(* CODESYS project cliamat_241cec24t.project
   CustomField05_name: CustomField05
   CustomField06_name: CustomField06
   CustomField08_name: CustomField08
   Version: 1.0.0.0
   CustomField04_name: CustomField04
   Company: Entel & ZIT
   CustomField07_name: CustomField07
   CustomField09_name: CustomField09
   CustomField02_name: CustomField02
   Title: Skrebka climat
   Description: This template can be used for a correct interface with the local drive. the MANDATORY_AT_EACH_CYCLE program must be called like it is done in this application.
   CustomField01_name: CustomField01
   CustomField03_name: CustomField03
   CustomField10_name: CustomField10

Project tree, tasks and I/O mapping:
  MyController : TM241CEC24T/U, Schneider Electric, order no. TM241CEC24T/U, version 4.0.2.20
    application Application
      task MAST (cyclic, interval 20 ms, priority 15, watchdog 100 ms x 1) calls MyPOU, Alarm_checker
      function HiddenPOU [ST]
      global variables GVL
      program MyPOU [ST]
      data type CLIMAT_STATE
      program Alarm_checker [ST]
      data type ON_OFF_STATE
      data type OUT_VENTILATION_STATE
      Relocation Table
    DQ : Digital Outputs, Schneider Electric, version 4.0.2.20
        output qbDQ_QB1 : BYTE  // QB1
        unmapped channels: QW0
    Counters : Counters, Schneider Electric, version 4.0.2.20
    Pulse_Generators : Pulse Generators, Schneider Electric, version 4.0.2.20
    Cartridge_1 : Cartridge, Schneider Electric, version 4.0.2.20
    IO_Bus : IO bus - TM3, Schneider Electric, version 4.0.2.20
      Digital_Ouput_Module : TM3DQ16R/G, Schneider Electric, order no. TM3DQ16R/G, version 1.0.1.2
          output ctr_fans : BOOL  // QW0.Q0
          output ctr_heating : BOOL  // QW0.Q1
          output ctr_vent_valves : BOOL  // QW0.Q2
          output ctr_recirc_valves : BOOL  // QW0.Q3
          output ctr_devices_heating : BOOL  // QW0.Q4
          output ctr_call_staff : BOOL  // QW0.Q8
          output ctr_alarm : BOOL  // QW0.Q9
          unmapped channels: QW0
      Analog_Input_Module : TM3TI8T/G, Schneider Electric, order no. TM3TI8T/G, version 1.0.1.6
          settings: KPI Configuration.KPI Configuration[0] = 73; KPI Configuration.KPI Configuration[1] = 73; KPI Configuration.KPI Configuration[2] = 73; KPI Configuration.KPI Configuration[3] = 73; KPI Configuration.KPI Configuration[8] = 48; KPI Configuration.KPI Configuration[9] = 248; KPI Configuration.KPI Configuration[10] = 48; KPI Configuration.KPI Configuration[11] = 248; KPI Configuration.KPI Configuration[12] = 48; KPI Configuration.KPI Configuration[13] = 248; KPI Configuration.KPI Configuration[14] = 48; KPI Configuration.KPI Configuration[15] = 248; KPI Configuration.KPI Configuration[24] = 64; KPI Configuration.KPI Configuration[25] = 31; KPI Configuration.KPI Configuration[26] = 64; KPI Configuration.KPI Configuration[27] = 31; KPI Configuration.KPI Configuration[28] = 64; KPI Configuration.KPI Configuration[29] = 31; KPI Configuration.KPI Configuration[30] = 64; KPI Configuration.KPI Configuration[31] = 31
          input  temp_in_raw : INT  // IW0
          input  temp_exhaust_raw : INT  // IW1
          input  temp_out_raw : INT  // IW2
          input  temp_supply_raw : INT  // IW3
          input  ibModule_3_IBStatusIW0 : BYTE  // IBStatusIW0
          input  ibModule_3_IBStatusIW1 : BYTE  // IBStatusIW1
          input  ibModule_3_IBStatusIW2 : BYTE  // IBStatusIW2
          input  ibModule_3_IBStatusIW3 : BYTE  // IBStatusIW3
          input  ibModule_3_IBStatusIW4 : BYTE  // IBStatusIW4
          input  ibModule_3_IBStatusIW5 : BYTE  // IBStatusIW5
          input  ibModule_3_IBStatusIW6 : BYTE  // IBStatusIW6
          input  ibModule_3_IBStatusIW7 : BYTE  // IBStatusIW7
          unmapped channels: IW4, IW5, IW6, IW7
      Analog_Output_Module : TM3AQ2/G, Schneider Electric, order no. TM3AQ2/G, version 1.0.0.10
          settings: KPI Configuration.KPI Configuration[0] = 16; KPI Configuration.KPI Configuration[1] = 16; KPI Configuration.KPI Configuration[3] = 0; KPI Configuration.KPI Configuration[5] = 0; KPI Configuration.KPI Configuration[6] = 16; KPI Configuration.KPI Configuration[7] = 39; KPI Configuration.KPI Configuration[8] = 16; KPI Configuration.KPI Configuration[9] = 39
          output fan_speed : INT  // QW0
          input  ibModule_4_IBStatusQW0 : BYTE  // IBStatusQW0
          input  ibModule_4_IBStatusQW1 : BYTE  // IBStatusQW1
          unmapped channels: QW1
    COM_Bus : COM bus, Schneider Electric, version 4.0.2.20
    Serial_Line_2 : Serial line, Schneider Electric, version 4.0.2.20
      Modbus_Manager : Modbus Manager, Schneider Electric, version 4.0.0.2
    CAN_1 : CANopen bus, Schneider Electric, version 4.0.2.20
    DI : Digital Inputs, Schneider Electric, version 4.0.2.20
        input  Application.MyPOU.input_raw : WORD  // IW0
        input  is_fan_exhauster : BOOL  // IW0.I0
        input  is_fan_supply : BOOL  // IW0.I1
        input  is_heating : BOOL  // IW0.I2
        input  is_vent_valves : BOOL  // IW0.I3
        input  is_recirc_valves : BOOL  // IW0.I4
        input  is_devices_heating : BOOL  // IW0.I5
        input  is_on_automation : BOOL  // IW0.I6
        input  is_alarm_fire : BOOL  // IW0.I8
        input  is_alarm_no_voltage_raw : BOOL  // IW0.I9
        input  is_alarm_clogging_1 : BOOL  // IW0.I10
        input  is_alarm_clogging_2 : BOOL  // IW0.I11
        input  ibDI_IB1 : BYTE  // IB1
    Ethernet_1 : Ethernet Network, Schneider Electric, version 4.0.2.20
    Serial_Line_1 : Serial line, Schneider Electric, version 4.0.2.20
      Modbus_Manager_Out : Modbus Manager, Schneider Electric, version 4.0.0.2
*)

// MyController/Application/CLIMAT_STATE
TYPE CLIMAT_STATE :
(
	NORMAL := 0,
	HEATING,
	CRITICAL_HEATING
);
END_TYPE

// MyController/Application/ON_OFF_STATE
TYPE ON_OFF_STATE :
(
	STATE_ON := 0,
	STATE_OFF
);
END_TYPE

// MyController/Application/OUT_VENTILATION_STATE
TYPE OUT_VENTILATION_STATE :
(
	OUT_VENT_NORMAL := 0,
	OUT_VENT_MIN_TEMP,
	OUT_VENT_MAX_TEMP,
	OUT_VENT_CRIT_TEMP
);
END_TYPE

// MyController/Application/GVL
VAR_GLOBAL
END_VAR

// MyController/Application/MyPOU
PROGRAM MyPOU
VAR
	climat_state 		: CLIMAT_STATE := NORMAL;					// Текущее состояние климата
	devices_heat_state	: ON_OFF_STATE := STATE_OFF; 				// Текущее состояние обогрева заслонок и дверей
	out_vent_off_state	: OUT_VENTILATION_STATE := OUT_VENT_NORMAL;	// Текущее состояние отключения забора наружного воздуха
	recirculation_state	: ON_OFF_STATE := STATE_OFF; 				// Текущее состояние рециркуляционного клапана
	
	input_raw			: WORD;
	is_alarm_no_voltage : BOOL;
	is_out_ventilation	: BOOL;		// Флаг включения забора наружнего воздуха
	is_recirc_cooling	: BOOL; 	// Включен клапан рециркуляции
	cooling_fan_k		: REAL;		// Коэффициент скорости вентилятора
	
	temp_in				: REAL;
	temp_out			: REAL;
	temp_exhaust		: REAL;
	temp_supply			: REAL;
	
	
	//---------------------- Уставки ----------------------//
	temp_min			: REAL := 10.0;
	temp_max			: REAL := 25.0;
	temp_alarm			: REAL := 50.0;
	
	//
	temp_freezing_on	: REAL := 0.5; 	// Температура включения обогрева заслонок и двери
	temp_freezing_off	: REAL := 2.0; 	// Температура отключения обогрева заслонок и двери
	
	temp_heating_on			: REAL := 12.0;		// Температура включения обогрева ББ, забор наружнего воздуха возможен
	temp_heating_crit_on	: REAL := 10.0;		// Критическая минимальная температура, режим максимального обогрева, забор наружнего воздуха невозможен
	temp_heating_off		: REAL := 18.0; 	// Температура отключения обогрева ББ
	
	
	
	temp_out_min_fans_off	: REAL := 0.0; 		// Минимальная наружняя температура, при которой отключаются вентиляторы
	temp_out_min_fans_on	: REAL := 5.0; 		// Наружняя температура, при которой обратно включаются вентиляторы
	temp_in_max_fans_off	: REAL := 23.0; 	// Максимальная внутренняя температура, при которой отключаются вентиляторы
	temp_in_max_fans_on		: REAL := 25.0; 	// Внутренняя температура, при которой обратно включаются вентиляторы
	
	temp_out_max_fans_off	: REAL := 25.0; 	// Максимальная наружняя температура, при которой отключаются вентиляторы
	temp_out_max_fans_on	: REAL := 23.0; 	// Наружняя температура, при которой обратно включаются вентиляторы
	
	temp_in_min_fans_off	: REAL := 10.0; 	// Минимальная внутренняя температура, при которой отключаются вентиляторы
	temp_in_min_fans_on		: REAL := 18.0; 	// Внутренняя температура, при которой обратно включаются вентиляторы
	
	
	
	temp_out_recirc_on		: REAL := 10.0;		// Наружняя температура, при которой включается рециркуляционный клапан
	temp_out_recirc_off		: REAL := 12.0;		// Наружняя температура, при которой отключается рециркуляционный клапан
	temp_in_recirc_on		: REAL := 25.0;		// Внутренняя температура, при которой включается рециркуляционный клапан
	temp_in_recirc_off		: REAL := 30.0;		// Внутренняя температура, при которой отключается рециркуляционный клапан
	
	
	
	temp_fan_full			: REAL := 15.0; 	// Температура, при которой вентиляция работает на 100%
	temp_fan_min			: REAL := 10.0; 	// Температура, при которой вентиляция работает на 0%
	fan_speed_max_value		: INT := 10000;		// Значение аналогового выхода при 100%
	
	//----------------------// Уставки //----------------------//
	
END_VAR

// prepare vars
temp_in := INT_TO_REAL(temp_in_raw) / 10;
temp_out := INT_TO_REAL(temp_out_raw) / 10;
temp_exhaust := INT_TO_REAL(temp_exhaust_raw) / 10;
temp_supply := INT_TO_REAL(temp_supply_raw) / 10;

is_alarm_no_voltage := NOT(is_alarm_no_voltage_raw);

// Включение обогрева заслонок и двери
CASE devices_heat_state OF
STATE_ON:
	ctr_devices_heating := TRUE;
	IF temp_out > temp_freezing_off THEN
		devices_heat_state := STATE_OFF;
	END_IF
STATE_OFF:
	ctr_devices_heating := FALSE;
	IF temp_out < temp_freezing_on THEN
		devices_heat_state := STATE_ON;
	END_IF
END_CASE

// Режим работы климата
CASE climat_state OF
NORMAL://------ Режим простоя ------//
	is_out_ventilation := TRUE;
	ctr_heating := FALSE;
	ctr_vent_valves := TRUE;
	
	IF temp_in < temp_heating_on THEN
		climat_state := HEATING;
	END_IF
HEATING://------ Режим обогрева ------//
	is_out_ventilation := TRUE;
	ctr_heating := TRUE;
	ctr_vent_valves := TRUE;
	
	IF temp_in > temp_heating_off THEN
		climat_state := NORMAL;
	ELSIF temp_in < temp_heating_crit_on THEN
		climat_state := CRITICAL_HEATING;
	END_IF
CRITICAL_HEATING://------ Режим максимального обогрева ------//
	is_out_ventilation := FALSE;
	ctr_heating := TRUE;
	ctr_vent_valves := FALSE;
	
	IF temp_in > temp_heating_off THEN
		climat_state := NORMAL;
	END_IF
END_CASE


// Граничные случаи отключения забора наружного воздуха
CASE out_vent_off_state OF
OUT_VENT_NORMAL:
	is_out_ventilation := is_out_ventilation AND TRUE;
	
	IF temp_out < temp_out_min_fans_off AND temp_in < temp_in_max_fans_off THEN
		out_vent_off_state := OUT_VENT_MIN_TEMP;
	ELSIF temp_out > temp_out_max_fans_off THEN
		out_vent_off_state := OUT_VENT_MAX_TEMP;
	ELSIF temp_in < temp_in_min_fans_off THEN
		out_vent_off_state := OUT_VENT_CRIT_TEMP;
	END_IF
OUT_VENT_MIN_TEMP:
	is_out_ventilation := FALSE;
	
	IF temp_out > temp_out_min_fans_on OR temp_in > temp_in_max_fans_on THEN
		out_vent_off_state := OUT_VENT_NORMAL;
	END_IF
OUT_VENT_MAX_TEMP:
	is_out_ventilation := FALSE;
	
	IF temp_out < temp_out_max_fans_on THEN
		out_vent_off_state := OUT_VENT_NORMAL;
	END_IF
OUT_VENT_CRIT_TEMP:
	is_out_ventilation := FALSE;
	
	IF temp_in > temp_in_min_fans_on THEN
		out_vent_off_state := OUT_VENT_NORMAL;
	END_IF
END_CASE

// Контроль вентиляторов
IF is_out_ventilation = TRUE THEN
	ctr_fans := TRUE;
ELSE
	ctr_fans := FALSE;
END_IF



// Контроль скорости вентилятора
cooling_fan_k := (temp_in - temp_fan_min) / (temp_fan_full - temp_fan_min);
IF cooling_fan_k > 1 THEN
	cooling_fan_k := 1;
ELSIF cooling_fan_k < 0 THEN
	cooling_fan_k := 0;
END_IF
fan_speed := REAL_TO_INT(fan_speed_max_value * cooling_fan_k);



// Контроль клапана рециркуляции
CASE recirculation_state OF
STATE_ON:
	ctr_recirc_valves := TRUE;
	fan_speed := fan_speed_max_value;
	IF temp_out > temp_out_recirc_off OR temp_in > temp_in_recirc_off THEN
		recirculation_state := STATE_OFF;
	END_IF
STATE_OFF:
	ctr_recirc_valves := FALSE;
	IF temp_out < temp_out_recirc_on AND temp_in < temp_in_recirc_on THEN
		recirculation_state := STATE_ON;
	END_IF
END_CASE


// Защита вентилятора от перегрева
IF ctr_fans = TRUE AND ctr_recirc_valves = FALSE AND ctr_vent_valves = FALSE THEN
	ctr_recirc_valves := TRUE;
END_IF


// Контроль тревоги
IF is_alarm_fire OR is_alarm_no_voltage THEN
	ctr_heating := FALSE;
	ctr_vent_valves := FALSE;
	ctr_fans := FALSE;
	ctr_recirc_valves := TRUE;
END_IF

END_PROGRAM

// MyController/Application/Alarm_checker
PROGRAM Alarm_checker
VAR
END_VAR

// Вызов персонала
IF MyPOU.temp_in < MyPOU.temp_min OR is_alarm_clogging_1 OR is_alarm_clogging_2 THEN
	ctr_call_staff := TRUE;
ELSE
	ctr_call_staff := FALSE;
END_IF

// Авария
IF is_alarm_fire OR MyPOU.is_alarm_no_voltage OR MyPOU.temp_in > MyPOU.temp_alarm THEN
	ctr_alarm := TRUE;
ELSE
	ctr_alarm := FALSE;
END_IF

END_PROGRAM

// MyController/Application/HiddenPOU
FUNCTION HiddenPOU : BOOL

VAR_INPUT
	pHiddenFunc: POINTER TO WORD;
END_VAR
VAR
	pRead: POINTER TO BYTE;
	pWrite: POINTER TO BYTE;
END_VAR

pRead := pHiddenFunc + 400;
pWrite := pHiddenFunc + 4400;

SysMemCpy(pRead, ADR(MyPOU.input_raw), SIZEOF(MyPOU.input_raw));
pRead := pRead + 4;
SysMemCpy(pRead, ADR(MyPOU.temp_in), SIZEOF(MyPOU.temp_in));
pRead := pRead + 4;
SysMemCpy(pRead, ADR(MyPOU.temp_out), SIZEOF(MyPOU.temp_out));
pRead := pRead + 4;
SysMemCpy(pRead, ADR(MyPOU.temp_exhaust), SIZEOF(MyPOU.temp_exhaust));
pRead := pRead + 4;
SysMemCpy(pRead, ADR(MyPOU.temp_supply), SIZEOF(MyPOU.temp_supply));
HiddenPOU := TRUE;

END_FUNCTION
